PROGRAM Error
VAR_INPUT

END_VAR
VAR
		i : INT;
	fbTest : FB_Test;
END_VAR

i := fbTest.Prop;

END_PROGRAM

(* stored: Version 1.1.0.1, ProductVersion 3.1.4024.12
   POU Error: Id {f73ef651-fb7d-41c1-b24f-41db580b875c}, SpecialFunc None *)
